# B&R Automation Studio project Lab2
Automation Studio 4.5.2.102

## Configuration SampleText

### Task classes (Cpu.sw)
```
Cyclic#1 (cycle 2000 us, tolerance 0 us):
  ncsdcctrl <- ncsdcctrl.prg
Cyclic#4:
  Program <- Program.prg
DataObjects: Acp10sys
NcDataObjects: acp10etxen <- acp10etxen.dob, gAxis01a <- gAxis01obj.gAxis01a.dob, gAxis01i <- gAxis01obj.gAxis01i.dob
Binaries: TCData, udbdef, ashwd, Role, User, sysconf, ashwac, asfw, arconfig, iomap, Acp10map, acp10cfg
Libraries: Acp10sdc, sys_lib, Runtime, asstring, Acp10man, Acp10par, NcGlobal, Acp10_MC, brsystem, AsBrStr, astime, fileio, powerlnk, asieccon, DriveLib
```

### Hardware
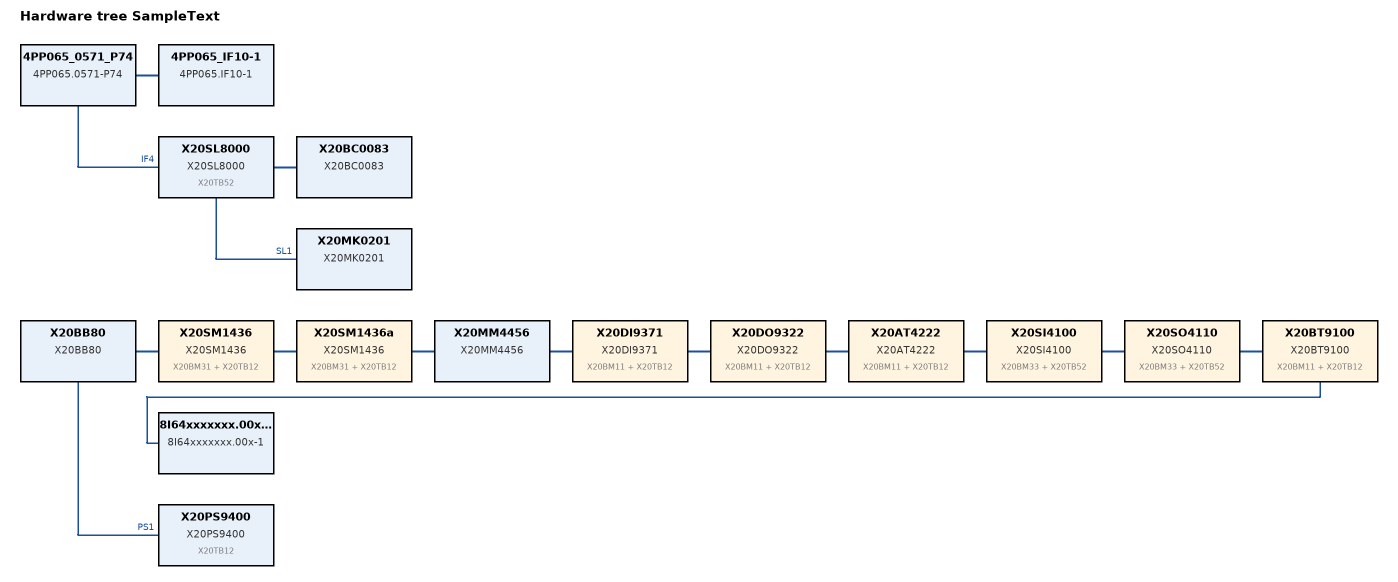
```
4PP065_0571_P74 : 4PP065.0571-P74 v1.1.2.0
  Connector IF4:
    EplInterfaceRedundant = 0
    EplEthInterfaceRedundant = 0
  Connector IF5:
    ActivateDevice = 1
    Mode = Manual
    InternetAddress = 10.0.1.9
    SubnetMask = 255.255.255.0
  ConfigurationID = labBR
  TimerDeviceType = EPLX2X
  TimerDevice = 4PP065_0571_P74.IF4
  TaskClassIdleTime = 2000
  Cyclic1Duration = 2000
  Cyclic1Tolerance = 0
  Cyclic1Output = 1
4PP065_IF10-1 : 4PP065.IF10-1 v1.0.3.0  [SS -> 4PP065_0571_P74.SS1]
8I64xxxxxxx.00x-1 : 8I64xxxxxxx.00x-1 v1.3.9.1  [X2X1 -> X20BT9100.X2X1 [Cable Type=X2XCable, Length=10, Version=1.0.0.2]]
  packedETAD = packed
  packedETI = packed
  packedCMDD = packed
  packedCMI = packed
X20AT4222 : X20AT4222 v1.2.3.0  [SS1 -> X20TB12e.SS; SL -> X20BM11c.SL1]
X20BB80 : X20BB80 v1.0.2.0
X20BC0083 : X20BC0083 v2.9.0.0  [PLK1 -> X20SL8000.PLK2 (NodeNumber=2) [Cable Type=PowerlinkCable, Length=10, Version=1.0.0.2]; SL -> X20BB80.SL1]
X20BM11 : X20BM11 v1.0.0.1  [X2X1 -> X20BM33a.X2X2]
X20BM11a : X20BM11 v1.0.0.1  [X2X1 -> X20MM4456.X2X2]
X20BM11b : X20BM11 v1.0.0.1  [X2X1 -> X20BM11a.X2X2]
X20BM11c : X20BM11 v1.0.0.1  [X2X1 -> X20BM11b.X2X2]
X20BM31 : X20BM31 v1.0.0.1  [X2X1 -> X20BB80.IF1]
X20BM31a : X20BM31 v1.0.0.1  [X2X1 -> X20BM31.X2X2]
X20BM33 : X20BM33 v1.0.0.4  [X2X1 -> X20BM11c.X2X2]
X20BM33a : X20BM33 v1.0.0.4  [X2X1 -> X20BM33.X2X2]
X20BT9100 : X20BT9100 v1.0.3.0  [SS1 -> X20TB12f.SS; SL -> X20BM11.SL1]
X20DI9371 : X20DI9371 v1.0.2.0  [SS1 -> X20TB12c.SS; SL -> X20BM11a.SL1]
X20DO9322 : X20DO9322 v1.0.3.0  [SS1 -> X20TB12d.SS; SL -> X20BM11b.SL1]
X20MK0201 : X20MK0201 v1.0.0.0  [SL -> X20SL8000.SL1]
X20MM4456 : X20MM4456 v1.1.5.0  [X2X1 -> X20BM31a.X2X2]
X20PS9400 : X20PS9400 v1.0.2.4  [SS1 -> X20TB12.SS; PS -> X20BB80.PS1]
X20SI4100 : X20SI4100 v1.10.1.1  [SS1 -> X20TB52.SS; SL -> X20BM33.SL1]
X20SL8000 : X20SL8000 v1.6.5.1  [PLK1 -> 4PP065_0571_P74.IF4 (NodeNumber=1) [Cable Type=PowerlinkCable, Length=10, Version=1.0.0.2]; PLK2 -> X20BC0083.PLK1 (NodeNumber=1) [Cable Type=PowerlinkCable, Length=10, Version=1.0.0.2]; SS1 -> X20TB52b.SS]
  SafeProject = SafeLOGIC-1
X20SM1436 : X20SM1436 v1.4.2.1  [SS1 -> X20TB12a.SS; SL -> X20BM31.SL1]
X20SM1436a : X20SM1436 v1.4.2.1  [SS1 -> X20TB12b.SS; SL -> X20BM31a.SL1]
X20SO4110 : X20SO4110 v1.10.1.1  [SS1 -> X20TB52a.SS; SL -> X20BM33a.SL1]
  SafeModuleID = 3
X20TB12 : X20TB12 v1.0.0.0
X20TB12a : X20TB12 v1.0.0.0
X20TB12b : X20TB12 v1.0.0.0
X20TB12c : X20TB12 v1.0.0.0
X20TB12d : X20TB12 v1.0.0.0
X20TB12e : X20TB12 v1.0.0.0
X20TB12f : X20TB12 v1.0.0.0
X20TB52 : X20TB52 v1.0.0.1
X20TB52a : X20TB52 v1.0.0.1
X20TB52b : X20TB52 v1.0.0.1
```

## Logical view

### Program Logical/Program (ANSIC)

#### Cyclic.c
```c
#include <bur/plctypes.h>

#ifdef _DEFAULT_INCLUDES
	#include <AsDefault.h>
#endif

void _CYCLIC ProgramCyclic(void)
{
	DoorStateMachine(&doorSM);
	ledSM.state = doorSM.state;
	LedStateMachine(&ledSM);

	stateMachine.speed = doorSM.speed;
	stateMachine.command = doorSM.speed != 0 ? CMD_SWITCH_ON : CMD_ENABLE;
	DriveStateMachine(&stateMachine);
}
```

### Library Logical/DriveLib (ANSIC)

#### Constants.var
```iecst
VAR CONSTANT
	SLOW_SPEED : UINT := 300;
	FAST_SPEED : UINT := 700;
END_VAR
```

#### DriveLib.fun
```iecst
{REDUND_ERROR} {REDUND_UNREPLICABLE} FUNCTION_BLOCK DriveStateMachine (*TODO: Add your comment here*) (*$GROUP=User,$CAT=User,$GROUPICON=User.png,$CATICON=User.png*)
	VAR_INPUT
		state : {REDUND_UNREPLICABLE} UINT;
		enable : {REDUND_UNREPLICABLE} BOOL;
	END_VAR
	VAR_OUTPUT
		speed : {REDUND_UNREPLICABLE} INT;
		command : {REDUND_UNREPLICABLE} UINT;
	END_VAR
END_FUNCTION_BLOCK

{REDUND_ERROR} {REDUND_UNREPLICABLE} FUNCTION_BLOCK LedStateMachine (*TODO: Add your comment here*) (*$GROUP=User,$CAT=User,$GROUPICON=User.png,$CATICON=User.png*)
	VAR_INPUT
		state : {REDUND_UNREPLICABLE} UINT;
	END_VAR
	VAR_OUTPUT
		led1 : {REDUND_UNREPLICABLE} BOOL;
		led2 : {REDUND_UNREPLICABLE} BOOL;
		led3 : {REDUND_UNREPLICABLE} BOOL;
		led4 : {REDUND_UNREPLICABLE} BOOL;
		timer : {REDUND_UNREPLICABLE} INT;
	END_VAR
END_FUNCTION_BLOCK

{REDUND_ERROR} {REDUND_UNREPLICABLE} FUNCTION_BLOCK DoorStateMachine (*TODO: Add your comment here*) (*$GROUP=User,$CAT=User,$GROUPICON=User.png,$CATICON=User.png*)
	VAR_INPUT
		state : {REDUND_UNREPLICABLE} UINT;
		sw1 : {REDUND_UNREPLICABLE} BOOL;
		sw2 : {REDUND_UNREPLICABLE} BOOL;
		sw3 : {REDUND_UNREPLICABLE} BOOL;
		sw4 : {REDUND_UNREPLICABLE} BOOL;
		direction : {REDUND_UNREPLICABLE} BOOL;
	END_VAR
	VAR_OUTPUT
		speed : {REDUND_UNREPLICABLE} INT;
	END_VAR
END_FUNCTION_BLOCK
```

#### DoorStateMachine.c
```c
#include <bur/plctypes.h>
#ifdef __cplusplus
	extern "C"
	{
#endif
	#include "DriveLib.h"
#ifdef __cplusplus
	};
#endif
/* TODO: Add your comment here */
void DoorStateMachine(struct DoorStateMachine* inst)
{
	switch(inst->state){
		case ST_INIT:
			break;
		case ST_UNKNOWN:
			if(inst->direction){
				inst->speed = -SLOW_SPEED;
				if(inst->sw4){
					setStateAndChangeSpeed(inst,ST_CLOSE);
				}
			}
			else{
				inst->speed = SLOW_SPEED;
				if(inst->sw1){
					setStateAndChangeSpeed(inst,ST_OPEN);
				}
			}
			break;
		case ST_OPEN:
			if(inst->direction){
				setStateAndChangeSpeed(inst,ST_ACC_NEG);
			}
			break;
		case ST_CLOSE:
			if(!inst->direction){
				setStateAndChangeSpeed(inst,ST_ACC_POS);
			}
			break;
		case ST_ACC_POS:
			if(inst->direction){
				setStateAndChangeSpeed(inst,ST_DEC_NEG);
			}
			else if(inst->sw3){
				setStateAndChangeSpeed(inst,ST_POS);
			}
			break;
		case ST_ACC_NEG:
			if(!inst->direction){
				setStateAndChangeSpeed(inst,ST_DEC_POS);
			}
			else if(inst->sw2){
				setStateAndChangeSpeed(inst,ST_NEG);
			}
			break;
		case ST_POS:
			if(inst->direction){
				setStateAndChangeSpeed(inst,ST_NEG);
			}
			else if(inst->sw2){
				setStateAndChangeSpeed(inst,ST_DEC_POS);
			}
			break;
		case ST_NEG:
			if(!inst->direction){
				setStateAndChangeSpeed(inst,ST_POS);
			}
			else if(inst->sw3){
				setStateAndChangeSpeed(inst,ST_DEC_NEG);
			}
			break;
		case ST_DEC_POS:
			if(inst->direction){
				setStateAndChangeSpeed(inst,ST_ACC_NEG);
			}
			else if(inst->sw1){
				setStateAndChangeSpeed(inst,ST_OPEN);
			}
			break;
		case ST_DEC_NEG:
			if(!inst->direction){
				setStateAndChangeSpeed(inst,ST_ACC_POS);
			}
			else if(inst->sw4){
				setStateAndChangeSpeed(inst,ST_CLOSE);
			}
			break;
		default:
			break;
	}
}

void setStateAndChangeSpeed(struct DoorStateMachine* inst, UINT state) {
	inst->state = state;
	switch(state){
		case ST_CLOSE:
			inst->speed = 0;
			break;
		case ST_OPEN:
			inst->speed = 0;
			break;
		case ST_ACC_POS:
			inst->speed = FAST_SPEED;
			break;
		case ST_DEC_POS:
			inst->speed = SLOW_SPEED;
			break;
		case ST_ACC_NEG:
			inst->speed = -FAST_SPEED;
			break;
		case ST_DEC_NEG:
			inst->speed = -SLOW_SPEED;
			break;
		default:
			break;
	}
}
```

#### DriveStateMachine.c
```c
#include <bur/plctypes.h>
#ifdef __cplusplus
	extern "C"
	{
#endif
	#include "DriveLib.h"
#ifdef __cplusplus
	};
#endif
/* TODO: Add your comment here */
void DriveStateMachine(struct DriveStateMachine* inst)
{
	if(inst->enable) {
		UINT stateMask = inst->state & 0x6f;
		switch (stateMask) {
			case ST_READY:
				inst->command = CMD_ENABLE;
				break;
			case ST_DISABLED:
				inst->command = CMD_SHUTDOWN;
				break;
			case ST_SWITCHED_ON:
				inst->command = CMD_SWITCH_ON;
		}
	}
	else
		inst->command = CMD_SHUTDOWN;
}
```

#### LedStateMachine.c
```c
#include <bur/plctypes.h>
#ifdef __cplusplus
	extern "C"
	{
#endif
	#include "DriveLib.h"
#ifdef __cplusplus
	};
#endif
/* TODO: Add your comment here */
void LedStateMachine(struct LedStateMachine* inst)
{
	switch(inst->state){
		case ST_UNKNOWN:
			if(inst->timer==10){
				setLeds(inst,!inst->led1,!inst->led1,!inst->led1,!inst->led1);
				inst->timer=0;
			}
			break;
		case ST_CLOSE:
			setLeds(inst,1,1,1,1);
			break;
		case ST_INIT:
		case ST_OPEN:
			setLeds(inst,0,0,0,0);
			break;
		case ST_ACC_POS:
		case ST_DEC_NEG:
			setLeds(inst,1,1,1,0);
			break;
		case ST_POS:
		case ST_NEG:
			setLeds(inst,1,1,0,0);
			break;
		case ST_DEC_POS:
		case ST_ACC_NEG:
			setLeds(inst,1,0,0,0);
			break;
	}
	inst->timer++;
}

void setLeds(struct LedStateMachine* inst, BOOL led1, BOOL led2, BOOL led3, BOOL led4){
	inst->led1 = led1;
	inst->led2 = led2;
	inst->led3 = led3;
	inst->led4 = led4;
}
```

Listed in the project but not available here: Logical/Global.typ, Logical/Global.var, Logical/Libraries, Logical/ncsdcctrl, Logical/acp10etxen, Logical/gAxis01obj
